Staubli VAL3: load.pgx

public program load(string x_sItem, num& i[])
begin
  // load the select trajctory
end
